TYPE DUT_STRUCT_LINECONTROLLER_PROD :
STRUCT
	sCellName			:STRING := 'LINECONTROLLER';
	sIpAddress			:STRING := '10.38.190.120';
	sAmsNetId			:STRING := '';
END_STRUCT
END_TYPE

(* stored: Version 1.1.0.1, ProductVersion 3.1.4024.6
   DUT DUT_STRUCT_LINECONTROLLER_PROD: Id {ff287891-1a46-4755-b5c5-c88f8f51062e} *)
